FUNCTION_BLOCK FB_Student

VAR
	sName : STRING := '';  // private — underscore convention
	sOutput : STRING := '';
	  nId : INT := 9; 
  
END_VAR
VAR_INPUT
	 nId1: INT :=343; 
END_VAR


VAR_OUTPUT
     nId2:INT := 32323;   // readable from outside
END_VAR

PROPERTY Id : INT
GET
Id := nId;
END_GET
SET
nId := Id;
END_SET
END_PROPERTY

PROPERTY Name : STRING
GET
//GET
Name := sName;
END_GET
SET
// SET
sName := Name;
END_SET
END_PROPERTY

END_FUNCTION_BLOCK

(* stored: Version 1.1.0.1, ProductVersion 3.1.4024.16
   POU FB_Student: Id {0893fcce-5e45-4b23-bd05-566cb9853b2f}, SpecialFunc None
   Property Id: Id {56f512ca-6eb2-40a2-bd5c-618ae51dadcb}
   Get Get: Id {be809445-f595-4307-abdb-f9b360bac18d}
   Set Set: Id {9c2c1e3e-6761-43c4-b70e-f5704f860063}
   Property Name: Id {bb3f729e-78f2-4d6d-b737-cdf37c6f4e1b}
   Get Get: Id {c125d67f-26eb-4e6d-856a-f05205e7debe}
   Set Set: Id {4e76c15a-5945-4ee4-ac3e-16e2d4410297} *)
